(*

.. <legal notes>

legal notes
=================
| SPDX-FileCopyrightText: © 2026 Oleksandr Tiutyk <trofimich@gmail.com>
| SPDX-License-Identifier: LGPL-3.0-only
| For details check: LGPL-3.0-only_

.. _LGPL-3.0-only: https://www.gnu.org/licenses/lgpl-3.0.en.html

.. </legal notes>

*)

{attribute 'no_explicit_call' := 'do not call this function block directly'} 
FUNCTION_BLOCK Operation EXTENDS Object IMPLEMENTS INamed
VAR
	{attribute 'hide'} 
	_ClassName : STRING := __POUNAME();
	
	{attribute 'hide'} 
	_Name : WSTRING;
END_VAR

{attribute 'monitoring' := 'call'}
PROPERTY ClassName : REFERENCE TO STRING
GET
ClassName REF= _ClassName;
END_GET
END_PROPERTY

METHOD FB_init : BOOL
VAR_INPUT
	(* if TRUE, the retain variables are initialized (warm start / cold start)*)
	bInitRetains	: BOOL;
	(* if TRUE, the instance afterwards gets moved into the copy code (online change)*)
	bInCopyCode	: BOOL;
	name : WSTRING;
END_VAR
_Name := name;
END_METHOD

{attribute 'monitoring' := 'call'}
PROPERTY FINAL Name : REFERENCE TO WSTRING
GET
Name REF= _Name;
END_GET
END_PROPERTY

{attribute 'monitoring' := 'call'}
PROPERTY NamespaceName : STRING
GET
NamespaceName := CurrentNamespace.Name;
END_GET
END_PROPERTY

{attribute 'monitoring' := 'call'}
PROPERTY SelfSize : ULINT
GET
SelfSize := XSIZEOF(THIS^);
END_GET
END_PROPERTY

END_FUNCTION_BLOCK

(* stored: Version 1.1.0.1
   POU Operation: Id {856aea8e-1241-4104-8feb-5476cb8fbca8}, SpecialFunc None
   Property ClassName: Id {3142e366-b89b-4444-b764-3f825bdc6d6a}
   Get Get: Id {b9a94c6b-1edf-4d76-af80-87d37d88f65f}
   Method FB_init: Id {a67d048a-93ef-4047-b96f-e73d16ee7e8e}
   Property Name: Id {03c97eee-32bf-4e2c-9c90-9e076a537e2f}
   Get Get: Id {8b41e209-52ce-40af-95c1-7b332322dbeb}
   Property NamespaceName: Id {263264a5-c98e-41b5-b8bb-05dda72b5bcd}
   Get Get: Id {1c29f2f5-90c5-4a3d-9532-19ff96ae710b}
   Property SelfSize: Id {39772ead-cc6e-4411-b576-e0b71a5afce1}
   Get Get: Id {4ab3c840-35da-42e6-8f34-5ae16131d9ce} *)
